// Mitsubishi GX Works2 project: PLC_Group31   PLC: FX3G

// global labels: Global1
VAR_GLOBAL
  X_7 AT X007 : BOOL;
  Y_10 AT Y007 : BOOL;
  X_5 AT X005 : BOOL;
  lemon AT D1100 : REAL;
  raspberry AT D1110 : REAL;
  stabilizer AT D1120 : REAL;
  gummy AT D1130 : REAL;
  initializeQuantity AT X007 : BOOL;
  X_1 AT X001 : BOOL;
END_VAR
VAR_GLOBAL CONSTANT
  constant0 : REAL;
END_VAR
VAR_GLOBAL
  Analoginput_1 AT D8280 : INT;
END_VAR
VAR_GLOBAL CONSTANT
  Divide : REAL := 400;
  Divide400 : REAL := 400;
END_VAR
VAR_GLOBAL
  GummyType AT D1145 : REAL;
END_VAR
VAR_GLOBAL CONSTANT
  constan1 : REAL := 1;
  constant5 : REAL := 5;
END_VAR
VAR_GLOBAL
  m_11 AT M11 : BOOL;
  m_17 AT M17 : BOOL;
END_VAR
VAR_GLOBAL CONSTANT
  constant6 : REAL := 6;
END_VAR
VAR_GLOBAL
  LemonIceCream AT D1150 : REAL;
  RaspberryIceCream AT D1160 : REAL;
END_VAR
VAR_GLOBAL CONSTANT
  constant40x7 : REAL := 280;
  constant65x7 : REAL := 455;
  constant15x7 : REAL := 105;
  constant55x7 : REAL := 385;
  constant95x7 : REAL := 665;
  constant30x7 : REAL := 210;
END_VAR
VAR_GLOBAL
  m_90 AT M90 : BOOL;
END_VAR
VAR_GLOBAL CONSTANT
  constan50x7 : REAL := 350;
  constant70x7 : REAL := 490;
END_VAR
VAR_GLOBAL
  m_24 AT M24 : BOOL;
  m_67 AT M67 : BOOL;
END_VAR
VAR_GLOBAL CONSTANT
  constan80x7 : REAL := 560;
END_VAR
VAR_GLOBAL
  Y_0 AT Y000 : BOOL;
  TC AT TC1 : BOOL;
END_VAR
VAR_GLOBAL CONSTANT
  IceCreamProcess : INT := 50;
  constant700 : REAL := 700;
END_VAR
VAR_GLOBAL
  X_2 AT X002 : BOOL;
  raspCooling AT D1345 : REAL;
  lemonCooling AT D1357 : REAL;
  m_55 AT M55 : BOOL;
END_VAR
VAR_GLOBAL CONSTANT
  Cooling : INT := 80;
END_VAR
VAR_GLOBAL
  tc_5 AT TC5 : BOOL;
  Y_2 AT Y002 : BOOL;
  x_3 AT X003 : BOOL;
  MixingTank AT D1456 : REAL;
  m_88 AT M88 : BOOL;
  Y_6 AT Y006 : BOOL;
  y_7 AT Y007 : BOOL;
  y_5 AT Y005 : BOOL;
  m_6 AT M6 : BOOL;
  ts_6 AT TS6 : BOOL;
  tc_6 AT TC6 : BOOL;
  m_96 AT M96 : BOOL;
  tc_7 AT TC7 : BOOL;
  ts_7 AT TS7 : BOOL;
END_VAR
VAR_GLOBAL CONSTANT
  three_sceonds : INT := 30;
END_VAR
VAR_GLOBAL
  timeAmount AT D3000 : INT;
END_VAR
VAR_GLOBAL CONSTANT
  five_sceonds : INT := 50;
END_VAR
VAR_GLOBAL
  TS_5 AT TS5 : BOOL;
  TS_1 AT TS1 : BOOL;
  TC_1 AT TC1 : BOOL;
  M_35 AT M35 : BOOL;
END_VAR
VAR_GLOBAL CONSTANT
  constant840 : REAL := 840;
END_VAR
VAR_GLOBAL
  m_92 AT M92 : BOOL;
  m_94 AT M94 : BOOL;
END_VAR
VAR_GLOBAL CONSTANT
  constant1260 : REAL := 1260;
END_VAR
VAR_GLOBAL
  TC_10 AT TC10 : BOOL;
  TS_10 AT TS10 : BOOL;
END_VAR
VAR_GLOBAL CONSTANT
  ConstHalfSec : INT := 2;
  constant4x7 : REAL := 28;
  constant10x7 : REAL := 70;
  constant10 : REAL := 10;
END_VAR
VAR_GLOBAL
  X_4 AT X004 : BOOL;
  BoxesQuantity : REAL;
  X_0 AT X000 : BOOL;
  M_101 : BOOL;
  Y_4 AT Y004 : BOOL;
  FirstCone AT CC9 : BOOL;
END_VAR
VAR_GLOBAL CONSTANT
  FirstConeee : INT := 1;
  ConesCounter7 : INT := 7;
END_VAR
VAR_GLOBAL
  ConesCounter AT CC8 : BOOL;
  first AT CS9 : BOOL;
  ConespackingDone AT CS8 : BOOL;
  packageCounter AT D3531 : REAL;
END_VAR
VAR_GLOBAL CONSTANT
  plusOne : REAL := 1;
END_VAR
VAR_GLOBAL
  M_105 AT M105 : BOOL;
END_VAR
VAR_GLOBAL CONSTANT
  Bit_0 : BOOL;
END_VAR
VAR_GLOBAL
  M_44 AT M44 : BOOL;
  M_40 AT M40 : BOOL;
  M_41 AT M41 : BOOL;
  M_42 AT M42 : BOOL;
  M_43 AT M43 : BOOL;
  M_1 AT M1 : BOOL;
END_VAR
VAR_GLOBAL CONSTANT
  outVal : INT := 40;
END_VAR
VAR_GLOBAL
  Analog_outputval AT D8282 : INT;
END_VAR

// task Task_01 (event TRUE, interval 0, priority 31): POU_01

PROGRAM POU_01
(* structured ladder/FBD written out as ST: instructions are called as NAME(EN, inputs, outputs); _pN, _eN, _tN stand for wires *)
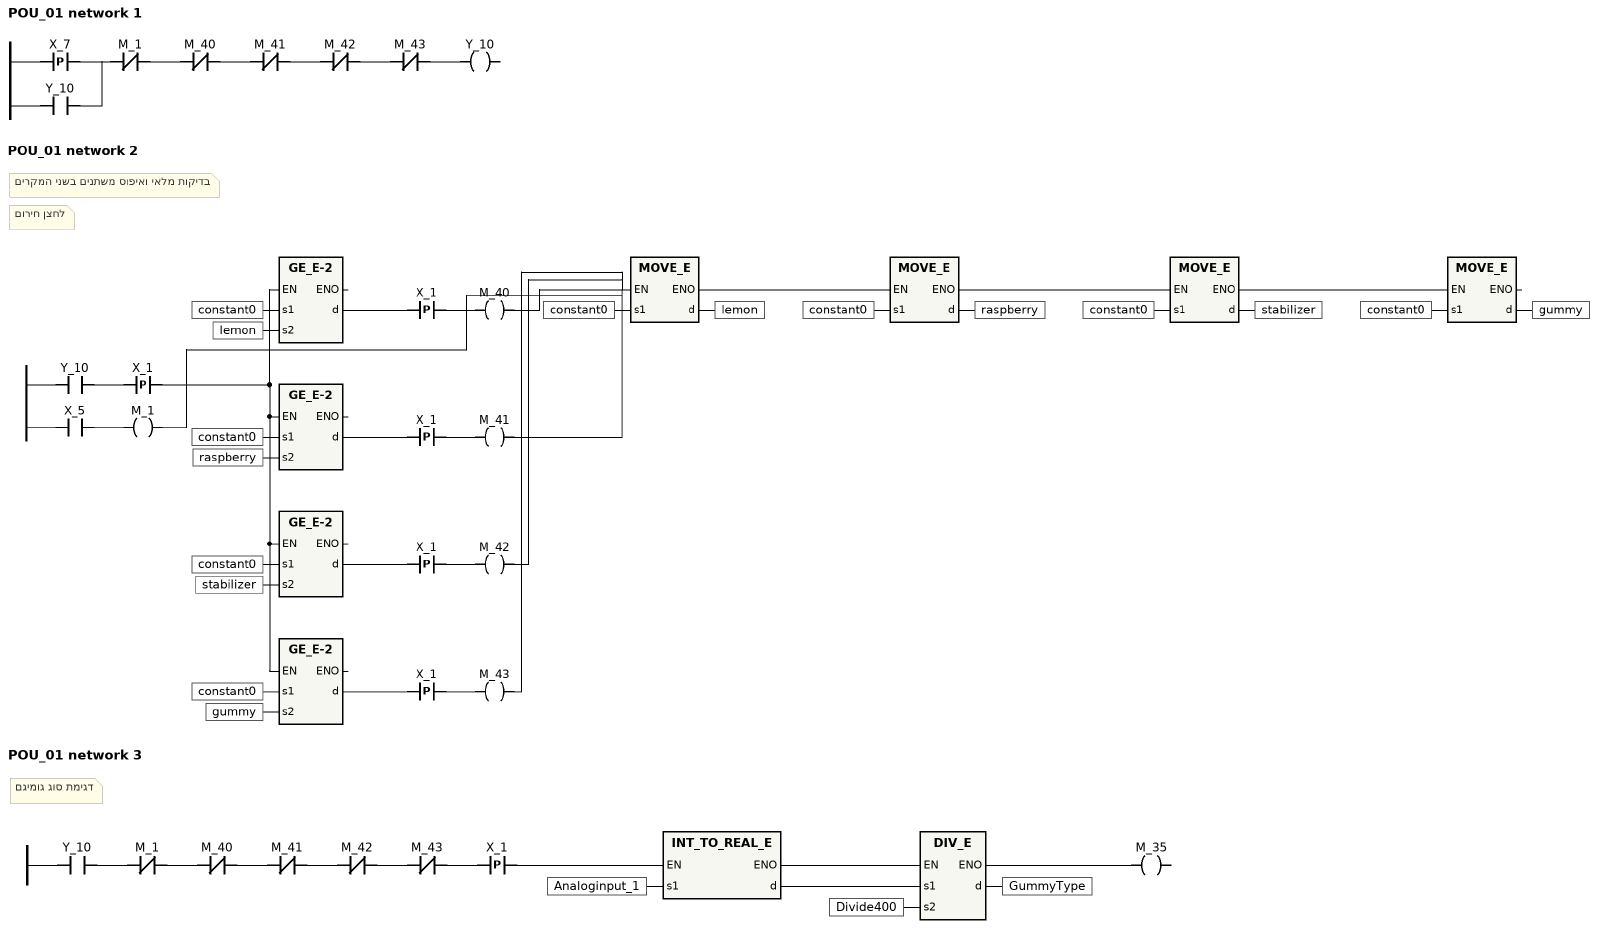
(* network 1 *)
Y_10 := (((((LDP(TRUE, X_7) OR Y_10) AND NOT M_1) AND NOT M_40) AND NOT M_41) AND NOT M_42) AND NOT M_43;
(* network 2 *)
(* בדיקות מלאי ואיפוס משתנים בשני המקרים *)
(* לחצן חירום *)
_p1 := Y_10 AND LDP(TRUE, X_1);
GE_E(_p1, constant0, lemon, _t2);
_p3 := _t2 AND LDP(TRUE, X_1);
M_40 := _p3;
GE_E(_p1, constant0, raspberry, _t4);
_p5 := _t4 AND LDP(TRUE, X_1);
M_41 := _p5;
GE_E(_p1, constant0, stabilizer, _t6);
_p7 := _t6 AND LDP(TRUE, X_1);
M_42 := _p7;
GE_E(_p1, constant0, gummy, _t8);
_p9 := _t8 AND LDP(TRUE, X_1);
M_43 := _p9;
M_1 := X_5;
_e10 := MOVE_E(_p3 OR _p5 OR _p7 OR _p9 OR X_5, constant0, lemon);
_e11 := MOVE_E(_e10, constant0, raspberry);
_e12 := MOVE_E(_e11, constant0, stabilizer);
MOVE_E(_e12, constant0, gummy);
(* network 3 *)
(* דגימת סוג גומיגם *)
_e2 := INT_TO_REAL_E(Y_10 AND NOT M_1 AND NOT M_40 AND NOT M_41 AND NOT M_42 AND NOT M_43 AND LDP(TRUE, X_1), Analoginput_1, _t1);
_e3 := DIV_E(_e2, _t1, Divide400, GummyType);
M_35 := _e3;
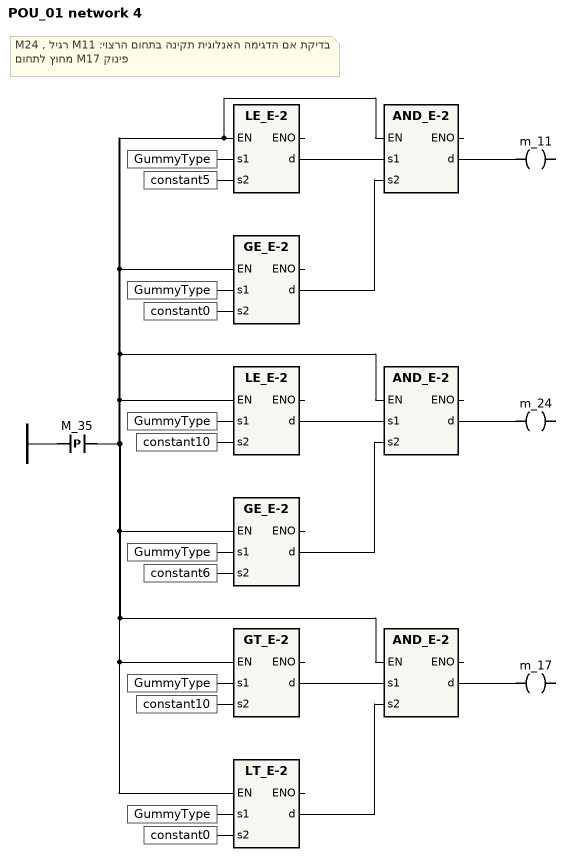
(* network 4 *)
(* בדיקת אם הדגימה האנלוגית תקינה בתחום הרצוי: M11 רגיל , M24 פינוק M17 מחוץ לתחום *)
_p1 := LDP(TRUE, M_35);
LE_E(_p1, GummyType, constant5, _t2);
GE_E(_p1, GummyType, constant0, _t3);
AND_E(_p1, _t2, _t3, _t4);
m_11 := _t4;
LE_E(_p1, GummyType, constant10, _t5);
GE_E(_p1, GummyType, constant6, _t6);
AND_E(_p1, _t5, _t6, _t7);
m_24 := _t7;
GT_E(_p1, GummyType, constant10, _t8);
LT_E(_p1, GummyType, constant0, _t9);
AND_E(_p1, _t8, _t9, _t10);
m_17 := _t10;
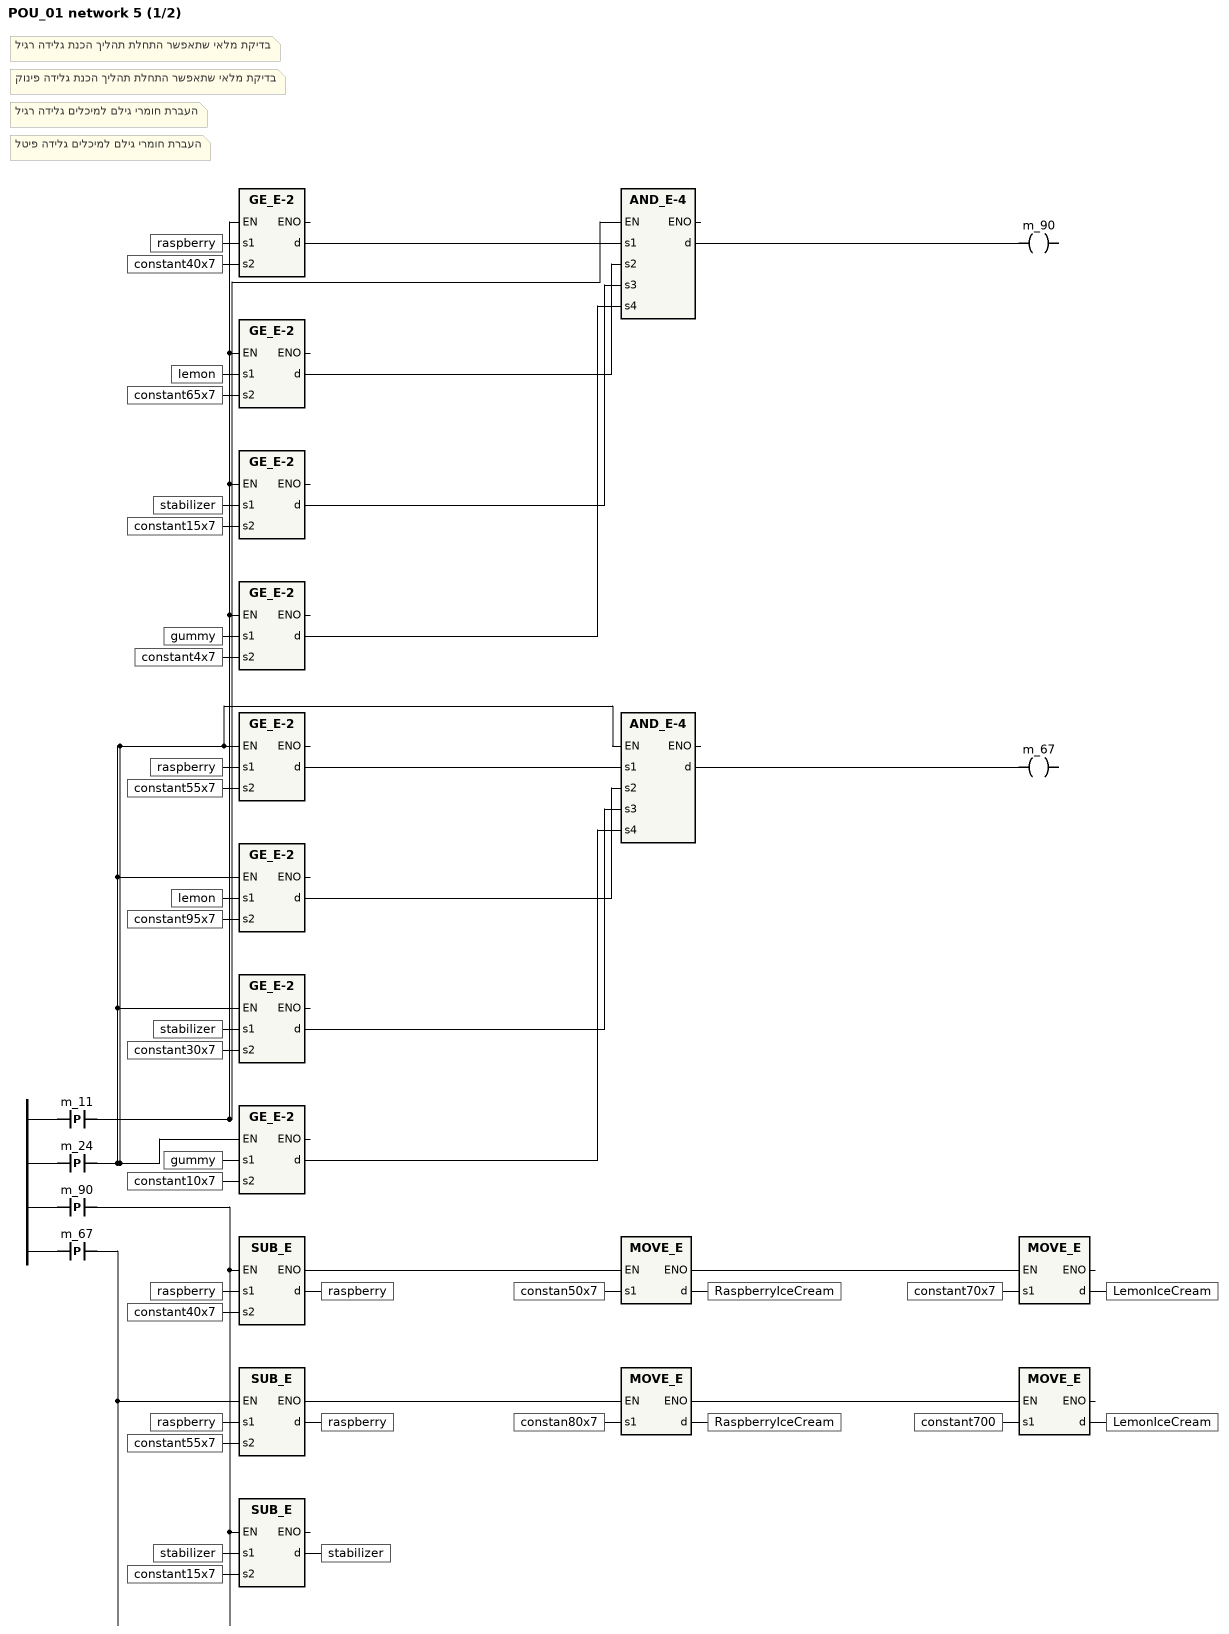
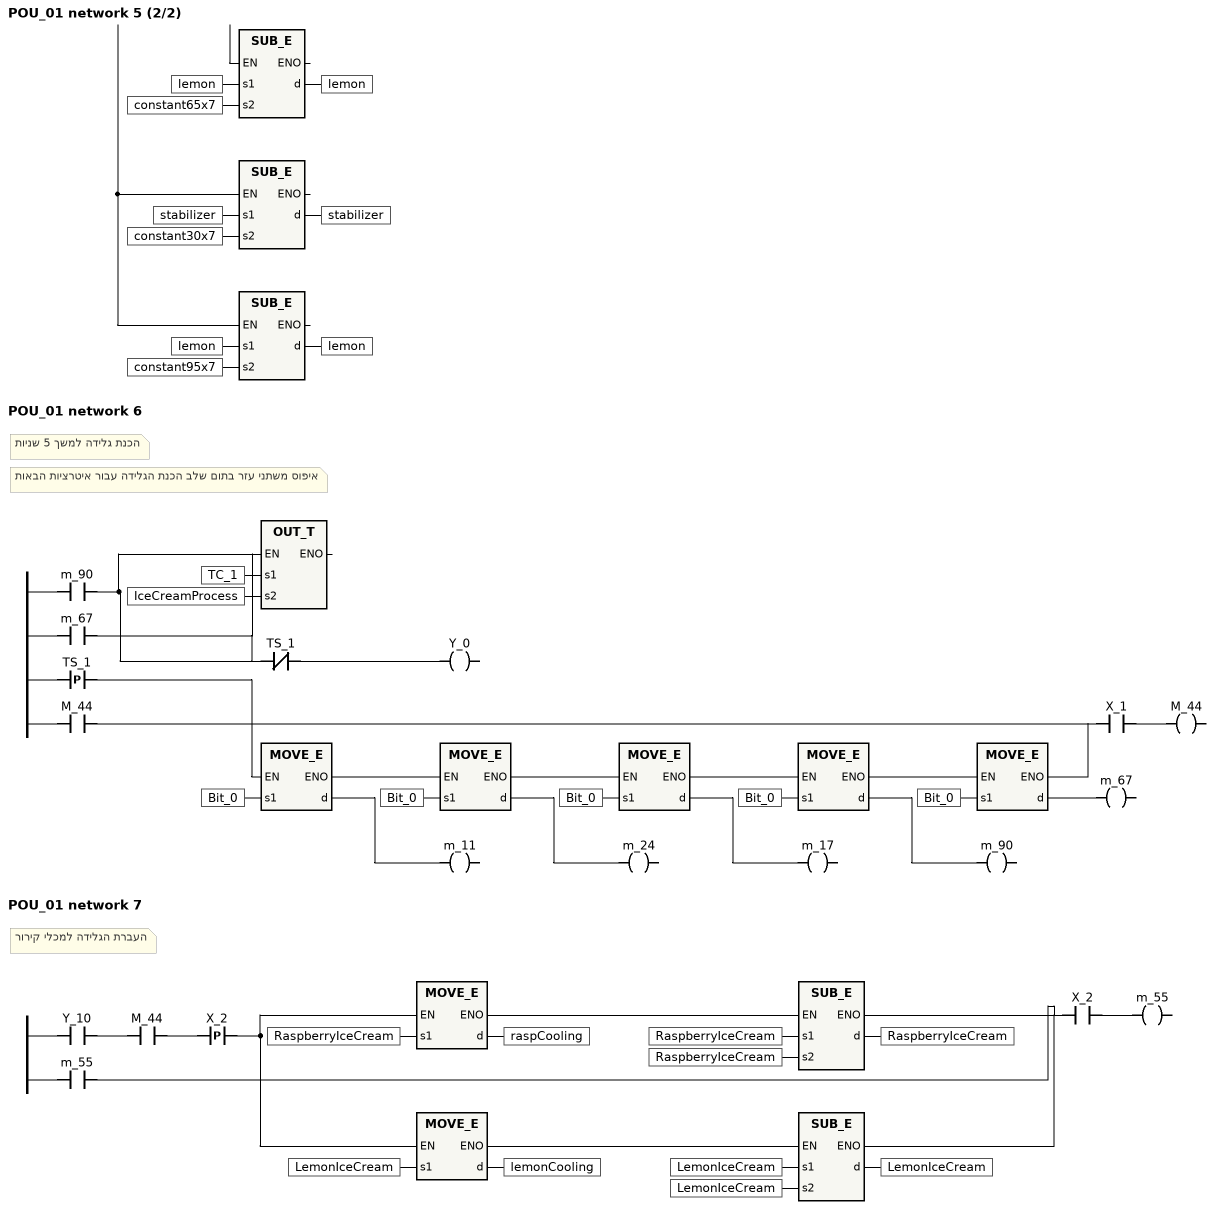
(* network 5 *)
(* בדיקת מלאי שתאפשר התחלת תהליך הכנת גלידה רגיל *)
(* בדיקת מלאי שתאפשר התחלת תהליך הכנת גלידה פינוק *)
(* העברת חומרי גילם למיכלים גלידה רגיל *)
(* העברת חומרי גילם למיכלים גלידה פיטל *)
_p1 := LDP(TRUE, m_11);
GE_E(_p1, raspberry, constant40x7, _t2);
GE_E(_p1, lemon, constant65x7, _t3);
GE_E(_p1, stabilizer, constant15x7, _t4);
GE_E(_p1, gummy, constant4x7, _t5);
AND_E(_p1, _t2, _t3, _t4, _t5, _t6);
m_90 := _t6;
_p7 := LDP(TRUE, m_24);
GE_E(_p7, raspberry, constant55x7, _t8);
GE_E(_p7, lemon, constant95x7, _t9);
GE_E(_p7, stabilizer, constant30x7, _t10);
GE_E(_p7, gummy, constant10x7, _t11);
AND_E(_p7, _t8, _t9, _t10, _t11, _t12);
m_67 := _t12;
_p13 := LDP(TRUE, m_90);
_e14 := SUB_E(_p13, raspberry, constant40x7, raspberry);
_e15 := MOVE_E(_e14, constan50x7, RaspberryIceCream);
MOVE_E(_e15, constant70x7, LemonIceCream);
SUB_E(_p13, stabilizer, constant15x7, stabilizer);
SUB_E(_p13, lemon, constant65x7, lemon);
_p16 := LDP(TRUE, m_67);
_e17 := SUB_E(_p16, raspberry, constant55x7, raspberry);
_e18 := MOVE_E(_e17, constan80x7, RaspberryIceCream);
MOVE_E(_e18, constant700, LemonIceCream);
SUB_E(_p16, stabilizer, constant30x7, stabilizer);
SUB_E(_p16, lemon, constant95x7, lemon);
(* network 6 *)
(* הכנת גלידה למשך 5 שניות *)
(* איפוס משתני עזר בתום שלב הכנת הגלידה עבור איטרציות הבאות *)
_p1 := m_90 OR m_67;
Y_0 := _p1 AND NOT TS_1;
OUT_T(_p1, TC_1, IceCreamProcess);
_e3 := MOVE_E(LDP(TRUE, TS_1), Bit_0, _t2);
_e5 := MOVE_E(_e3, Bit_0, _t4);
_e7 := MOVE_E(_e5, Bit_0, _t6);
_e9 := MOVE_E(_e7, Bit_0, _t8);
_e11 := MOVE_E(_e9, Bit_0, _t10);
M_44 := (_e11 OR M_44) AND X_1;
m_11 := _t2;
m_24 := _t4;
m_17 := _t6;
m_90 := _t8;
m_67 := _t10;
(* network 7 *)
(* העברת הגלידה למכלי קירור *)
_p1 := Y_10 AND M_44 AND LDP(TRUE, X_2);
_e2 := MOVE_E(_p1, RaspberryIceCream, raspCooling);
_e3 := SUB_E(_e2, RaspberryIceCream, RaspberryIceCream, RaspberryIceCream);
_e4 := MOVE_E(_p1, LemonIceCream, lemonCooling);
_e5 := SUB_E(_e4, LemonIceCream, LemonIceCream, LemonIceCream);
m_55 := (_e3 OR _e5 OR m_55) AND X_2;
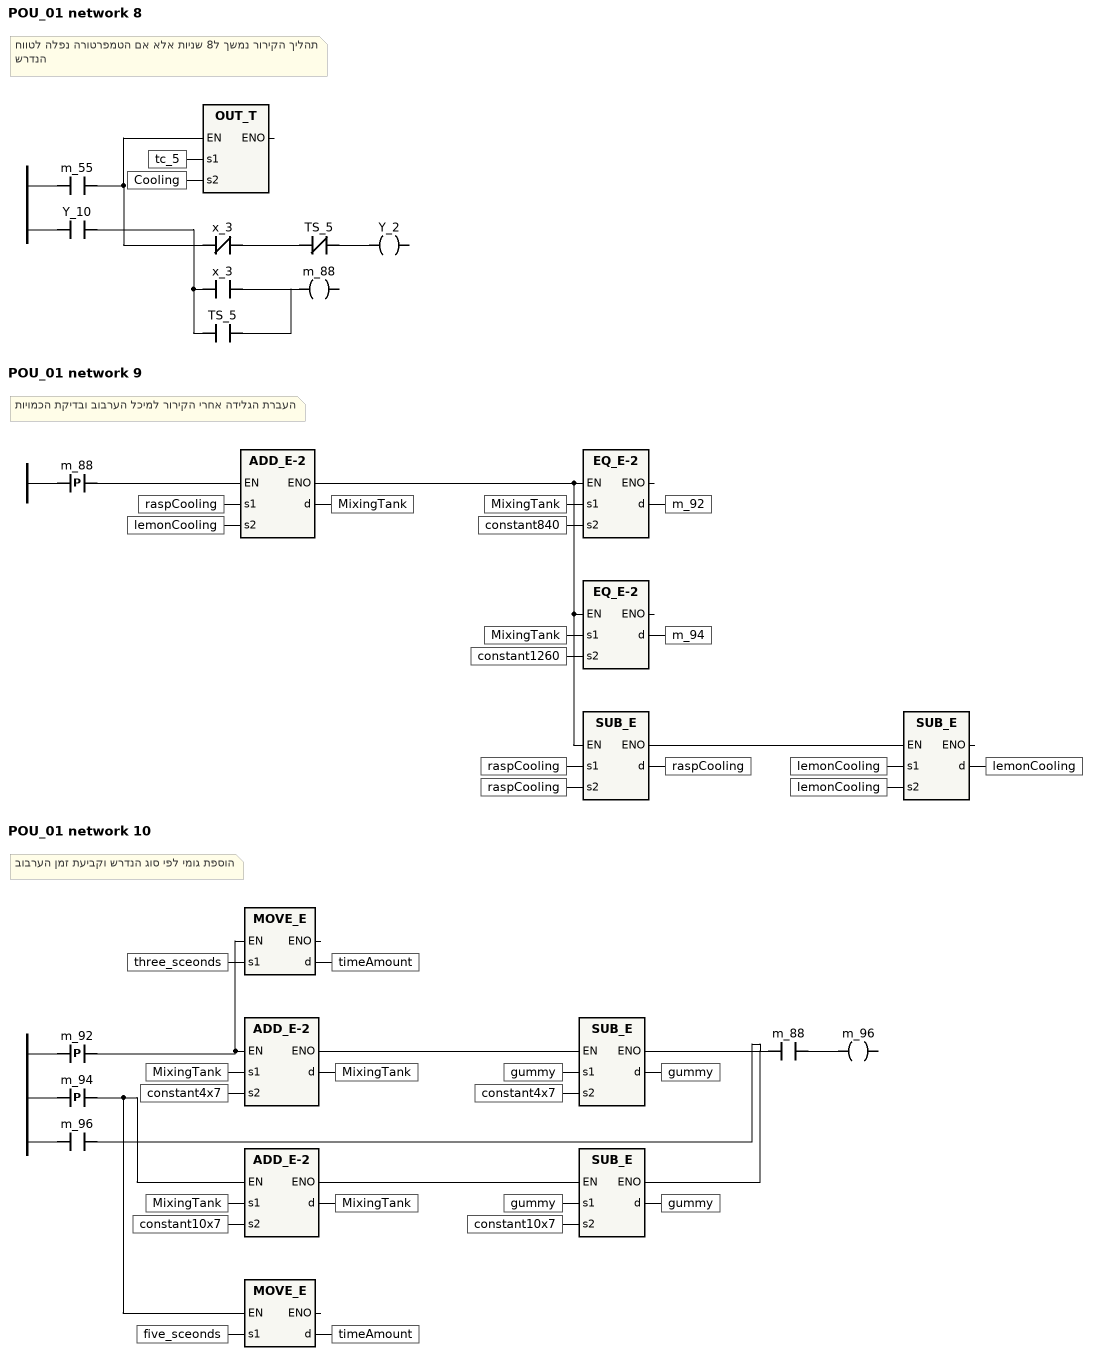
(* network 8 *)
(* תהליך הקירור נמשך ל8 שניות אלא אם הטמפרטורה נפלה לטווח הנדרש *)
Y_2 := m_55 AND NOT x_3 AND NOT TS_5;
OUT_T(m_55, tc_5, Cooling);
m_88 := (Y_10 AND x_3) OR (Y_10 AND TS_5);
(* network 9 *)
(* העברת הגלידה אחרי הקירור למיכל הערבוב ובדיקת הכמויות *)
_e1 := ADD_E(LDP(TRUE, m_88), raspCooling, lemonCooling, MixingTank);
EQ_E(_e1, MixingTank, constant840, m_92);
EQ_E(_e1, MixingTank, constant1260, m_94);
_e2 := SUB_E(_e1, raspCooling, raspCooling, raspCooling);
SUB_E(_e2, lemonCooling, lemonCooling, lemonCooling);
(* network 10 *)
(* הוספת גומי לפי סוג הנדרש וקביעת זמן הערבוב *)
_p1 := LDP(TRUE, m_92);
MOVE_E(_p1, three_sceonds, timeAmount);
_e2 := ADD_E(_p1, MixingTank, constant4x7, MixingTank);
_e3 := SUB_E(_e2, gummy, constant4x7, gummy);
_p4 := LDP(TRUE, m_94);
MOVE_E(_p4, five_sceonds, timeAmount);
_e5 := ADD_E(_p4, MixingTank, constant10x7, MixingTank);
_e6 := SUB_E(_e5, gummy, constant10x7, gummy);
m_96 := (_e3 OR _e6 OR m_96) AND m_88;
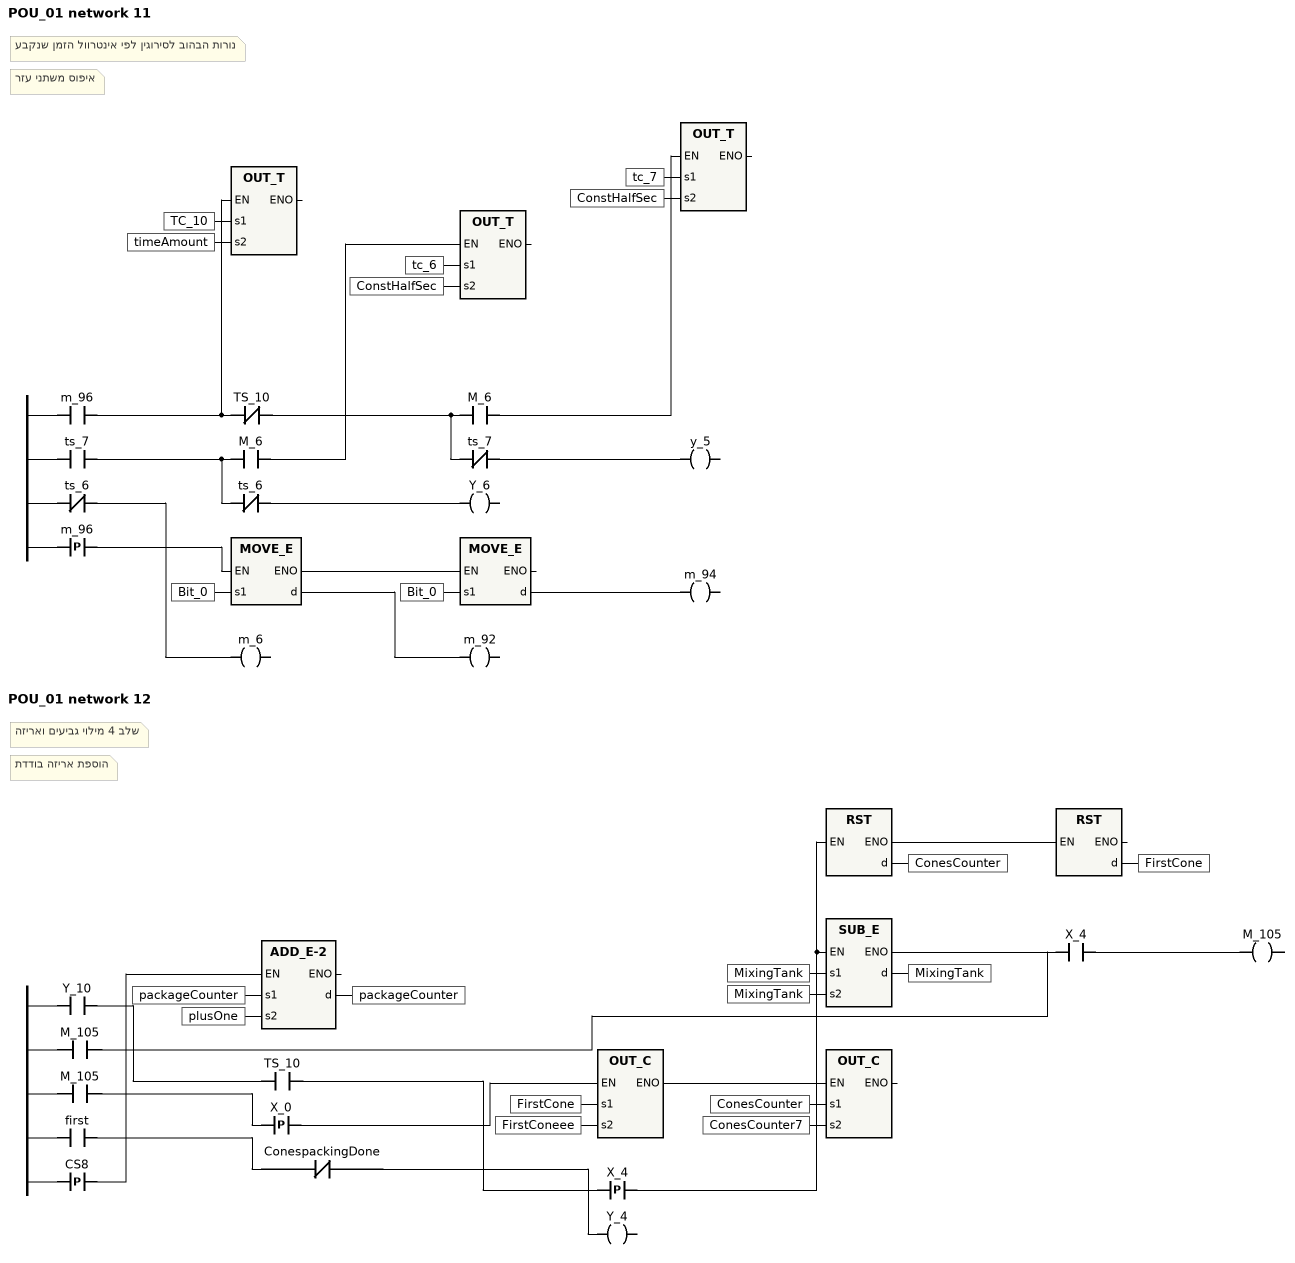
(* network 11 *)
(* נורות הבהוב לסירוגין לפי אינטרוול הזמן שנקבע *)
(* איפוס משתני עזר *)
_p1 := m_96 AND NOT TS_10;
OUT_T(_p1 AND M_6, tc_7, ConstHalfSec);
OUT_T(m_96, TC_10, timeAmount);
y_5 := _p1 AND NOT ts_7;
OUT_T(ts_7 AND M_6, tc_6, ConstHalfSec);
Y_6 := ts_7 AND NOT ts_6;
m_6 := NOT ts_6;
_e3 := MOVE_E(LDP(TRUE, m_96), Bit_0, _t2);
MOVE_E(_e3, Bit_0, _t4);
m_92 := _t2;
m_94 := _t4;
(* network 12 *)
(* שלב 4 מילוי גביעים ואריזה *)
(* הוספת אריזה בודדת *)
_p1 := Y_10 AND TS_10 AND LDP(TRUE, X_4);
_e2 := RST(_p1, ConesCounter);
RST(_e2, FirstCone);
_e3 := SUB_E(_p1, MixingTank, MixingTank, MixingTank);
M_105 := (_e3 OR M_105) AND X_4;
_e4 := OUT_C(M_105 AND LDP(TRUE, X_0), FirstCone, FirstConeee);
OUT_C(_e4, ConesCounter, ConesCounter7);
Y_4 := first AND NOT ConespackingDone;
ADD_E(LDP(TRUE, CS8), packageCounter, plusOne, packageCounter);
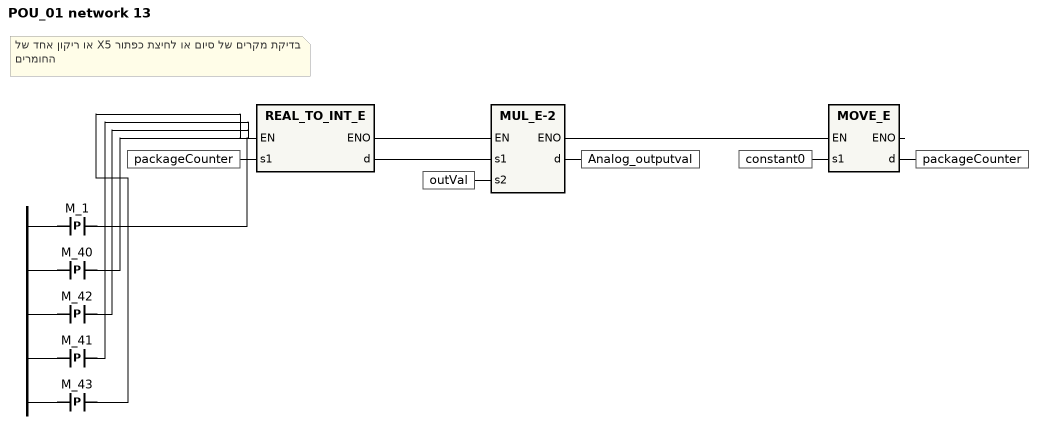
(* network 13 *)
(* בדיקת מקרים של סיום או לחיצת כפתור X5 או ריקון אחד של החומרים *)
_e2 := REAL_TO_INT_E(LDP(TRUE, M_1) OR LDP(TRUE, M_40) OR LDP(TRUE, M_42) OR LDP(TRUE, M_41) OR LDP(TRUE, M_43), packageCounter, _t1);
_e3 := MUL_E(_e2, _t1, outVal, Analog_outputval);
MOVE_E(_e3, constant0, packageCounter);
END_PROGRAM
